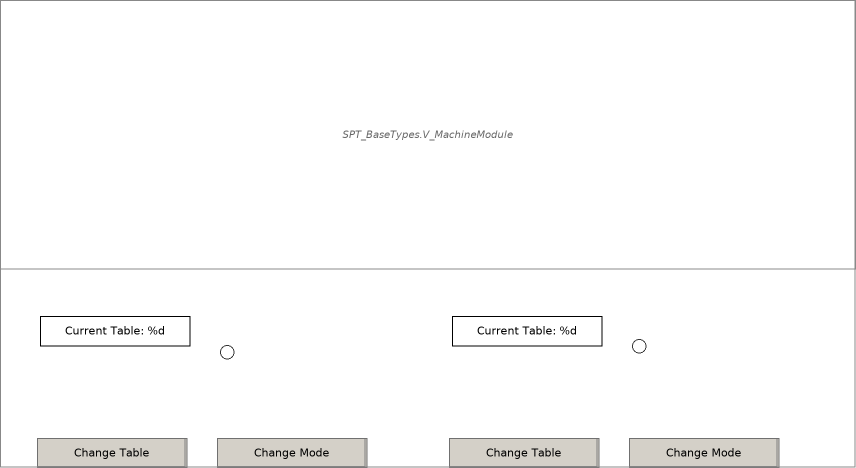
VISUALIZATION Visualization  // 856x468
    Frame (0,0 856x269)
        shows SPT_BaseTypes.V_MachineModule(HMI := MAIN.Machine.PackMLBaseModule_HMI)
    Button (37,438 150x30), "Change Table"
        toggle MAIN.Machine.CamModule_TableSelect.HMI.Cmd.ChangeTable
    Rectangle (40,316 150x30), "Current Table: %d", text variable: MAIN.Machine.CamModule_TableSelect.HMI.Sts.CurrentTable
    RadioButton (218,296 150x112), variable: MAIN.Machine.CamModule_TableSelect.HMI.Cfg.CamActivationMode
        Areas[0]: Text=Instantaneous
        Areas[1]: Text=Next Cycle
        Areas[2]: Text=As Soon As Possible
    Button (217,438 150x30), "Change Mode"
        toggle MAIN.Machine.CamModule_TableSelect.HMI.Cmd.ChangeMode
    Button (449,438 150x30), "Change Table"
        toggle MAIN.Machine.CamModule_UpdateTable.HMI.Cmd.ChangeTable
    Rectangle (452,316 150x30), "Current Table: %d", text variable: MAIN.Machine.CamModule_UpdateTable.HMI.Sts.CurrentTable
    RadioButton (630,296 150x100), variable: MAIN.Machine.CamModule_UpdateTable.HMI.Cfg.CamActivationMode
        Areas[0]: Text=Instantaneous
        Areas[1]: Text=Next Cycle
        Areas[2]: Text=As Soon As Possible
    Button (629,438 150x30), "Change Mode"
        toggle MAIN.Machine.CamModule_UpdateTable.HMI.Cmd.ChangeMode
END_VISUALIZATION

(* stored: Version 1.1.0.1, ProductVersion 3.1.4026.13
   Visu Visualization: Id {dcda8cdc-31c0-441c-9c53-44fba7b7ab38} *)
